FUNCTION_BLOCK FB_Standard_stuff
VAR_INPUT
	Bits_from_hmi:ARRAY[0..1] OF WORD;
	Creep_switch:BOOL;
	Slow_switch:BOOL;
	Normal_switch:BOOL;
	Watchdog_heartbeat:BOOL;
	System_start:BOOL;
	System_stop:BOOL;
	System_started:BOOL;
	SCC:BOOL;
END_VAR
VAR_OUTPUT
	Bits_to_hmi:ARRAY[0..1] OF WORD;
	Hmi_test_trip:BOOL;
	Watchdog_test_0:BOOL;
	Watchdog_test_1:BOOL;
	Activity:BOOL;
END_VAR

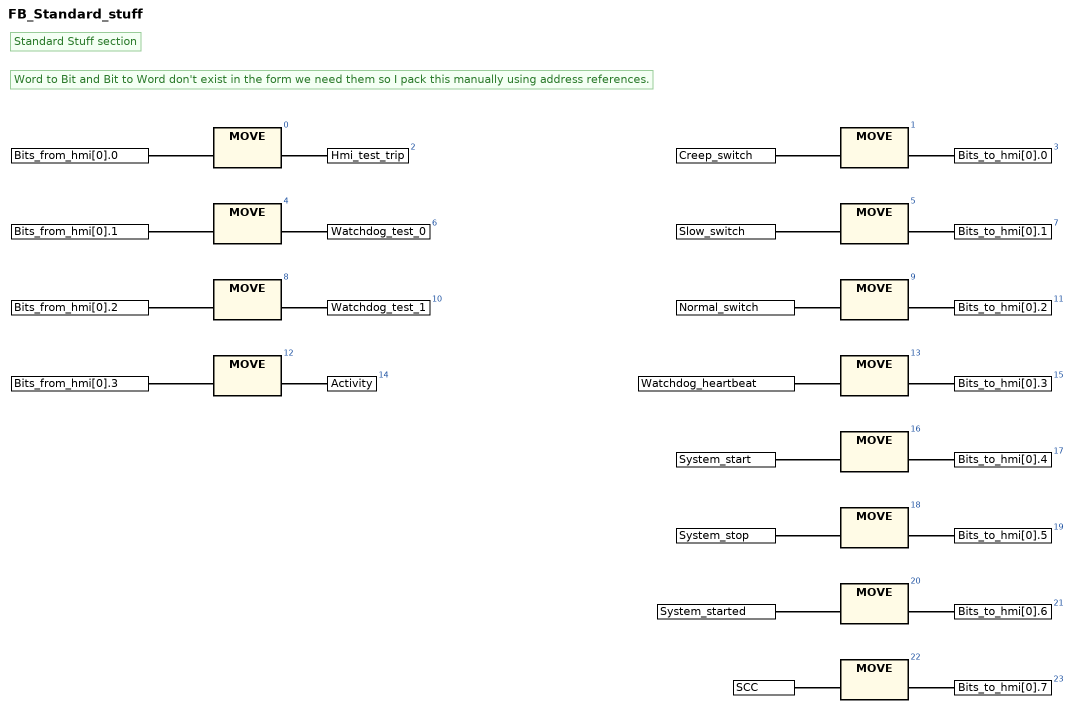
// Standard Stuff section
// Word to Bit and Bit to Word don't exist in the form we need them so I pack this manually using address references.
Hmi_test_trip := Bits_from_hmi[0].0;
Bits_to_hmi[0].0 := Creep_switch;
Watchdog_test_0 := Bits_from_hmi[0].1;
Bits_to_hmi[0].1 := Slow_switch;
Watchdog_test_1 := Bits_from_hmi[0].2;
Bits_to_hmi[0].2 := Normal_switch;
Activity := Bits_from_hmi[0].3;
Bits_to_hmi[0].3 := Watchdog_heartbeat;
Bits_to_hmi[0].4 := System_start;
Bits_to_hmi[0].5 := System_stop;
Bits_to_hmi[0].6 := System_started;
Bits_to_hmi[0].7 := SCC;

END_FUNCTION_BLOCK

(* stored: Version 1.1.0.1, ProductVersion 3.1.4024.0
   POU FB_Standard_stuff: Id {4cc38c31-b175-43ff-8b69-fa30cceab370}, SpecialFunc None *)
